{attribute addProperty BoxType "CU2508-0000-0017"}
{attribute addProperty Id "EPM_Inputs_ChannelAT %I*ARRAY[0..18] OF EPM_Inputs_Channel_7B63A807160200WcStateAT %I*WcState_98A4DF7520.250InfoDataAT %I*InfoData_BC63D37F80100"}
{attribute addProperty CRC "2816817870"}
{attribute addProperty SizeInBites "242"}
{attribute addProperty SizeInBytes "30.25"}
TYPE CU2508_36DE2952 :
STRUCT
	{attribute addProperty Name "EPM_Inputs_Channel"}
	EPM_Inputs_Channel : ARRAY[0..18] OF EPM_Inputs_Channel_7B63A807;
	{attribute addProperty Name "WcState"}
	WcState : WcState_98A4DF75;
	{attribute addProperty Name "InfoData"}
	InfoData : InfoData_BC63D37F;
END_STRUCT
END_TYPE

(* stored: Version 1.2.0.0, ProductVersion 3.1.4024.9
   DUT CU2508_36DE2952: Id {6051e168-32c5-4b9d-862d-8fda172eaac5} *)
